INTERFACE I_ManualUi

METHOD PUBLIC M_SetStateObject : BOOL
VAR_IN_OUT
	stStateObjectRef : ST_Object_Item;
END_VAR
END_METHOD

PROPERTY Name : ST_Text
GET
END_GET
END_PROPERTY

PROPERTY ObjectIndex : DINT
GET
END_GET
SET
END_SET
END_PROPERTY

END_INTERFACE

(* stored: Version 1.1.0.1, ProductVersion 3.1.4024.12
   Itf I_ManualUi: Id {001e1cb9-18f1-4c1b-87c0-1def144f453a}
   Method M_SetStateObject: Id {533965c2-f4bd-45d2-bd03-a27d7af9f40e}
   Property Name: Id {8fb561b9-b27e-446a-baba-602476846166}
   Get Get: Id {634b333d-76ac-43d2-a313-972a9501081b}
   Property ObjectIndex: Id {3d080eaa-5ac0-4d9f-815c-2d67188a0217}
   Get Get: Id {2cc7e4b1-b74a-4e2f-99a6-fc2f40eec5eb}
   Set Set: Id {e893e6b9-fc8b-40db-9c99-58664512ce60} *)
